/// MODULE INTERFACE INPUT AND OUTPUT 
TYPE DUT_MODULE_INTERFACE :
STRUCT
	///Information that the module reads
	Input: DUT_MODULE_INTERFACE_INPUT;
	///Information that the module write
	Output: DUT_MODULE_INTERFACE_OUTPUT;
END_STRUCT
END_TYPE

(* stored: Version 1.1.0.1, ProductVersion 3.1.0.25
   DUT DUT_MODULE_INTERFACE: Id {55e99faa-9e83-454e-84cc-bb9d737f7711} *)
